(* IEC 61131-3 sources: RL_MAR/experiments/comparison/llm4plc/results/gpt-4o_20260507_114630/20260507_120848, 4 files *)

(* ---- generated_code_iteration_0.st ---- *)
plaintext
START_ST
FUNCTION_BLOCK FB_CourseDifferenceControl
VAR_INPUT
    KOMPASS_GRAD : INT; // Compass heading in tenths of a degree
    KURS         : INT; // Desired course in tenths of a degree
END_VAR
VAR_OUTPUT
    KURS_DIFF    : INT; // Computed course difference in tenths of a degree
END_VAR
VAR
    temp_diff    : INT; // Temporary variable for intermediate calculations
END_VAR

// Logic for course difference computation
IF KOMPASS_GRAD < 0 THEN
    KURS_DIFF := 0; // Set output to 0 if KOMPASS_GRAD is less than 0
ELSE
    temp_diff := KURS - KOMPASS_GRAD; // Calculate the initial difference
    IF temp_diff > 1800 THEN
        KURS_DIFF := temp_diff - 3600; // Adjust if the difference is greater than 1800
    ELSIF temp_diff < -1800 THEN
        KURS_DIFF := temp_diff + 3600; // Adjust if the difference is less than -1800
    ELSE
        KURS_DIFF := temp_diff; // No adjustment needed
    END_IF;
END_IF;

END_FUNCTION_BLOCK

PROGRAM MAIN
VAR
    fbCourseDifferenceControl : FB_CourseDifferenceControl; // Instance of the function block
    KOMPASS_GRAD_MAIN         : INT; // Compass heading input
    KURS_MAIN                 : INT; // Desired course input
    KURS_DIFF_MAIN            : INT; // Output course difference
END_VAR

// Initialize input variables
KOMPASS_GRAD_MAIN := 0; // Example initialization, can be replaced with actual values
KURS_MAIN := 0;         // Example initialization, can be replaced with actual values

// Call the function block
fbCourseDifferenceControl(KOMPASS_GRAD := KOMPASS_GRAD_MAIN, KURS := KURS_MAIN);

// Retrieve the output from the function block
KURS_DIFF_MAIN := fbCourseDifferenceControl.KURS_DIFF;

END_PROGRAM
END_ST

(* ---- generated_code_iteration_1.st ---- *)
START_REASON
The validation feedback indicates that the `MAIN` program cannot be instantiated in CODESYS. This error occurs because in Structured Text (ST), a `PROGRAM` type cannot be instantiated like a `FUNCTION_BLOCK`. Instead, the `PROGRAM` type is executed directly as part of the PLC cycle. The issue arises from attempting to create an instance of the `MAIN` program, which is not allowed.

To resolve this, the `PROGRAM MAIN` section should be modified to directly execute the logic without attempting to instantiate it. The `FUNCTION_BLOCK FB_CourseDifferenceControl` is correctly implemented and can be used within the `PROGRAM MAIN` by directly invoking its logic.

Additionally, the initialization of input variables and the retrieval of output variables should be adjusted to align with the corrected structure.

END_REASON

START_ST
FUNCTION_BLOCK FB_CourseDifferenceControl
VAR_INPUT
    KOMPASS_GRAD : INT; // Compass heading in tenths of a degree
    KURS         : INT; // Desired course in tenths of a degree
END_VAR
VAR_OUTPUT
    KURS_DIFF    : INT; // Computed course difference in tenths of a degree
END_VAR
VAR
    temp_diff    : INT; // Temporary variable for intermediate calculations
END_VAR

// Logic for course difference computation
IF KOMPASS_GRAD < 0 THEN
    KURS_DIFF := 0; // Set output to 0 if KOMPASS_GRAD is less than 0
ELSE
    temp_diff := KURS - KOMPASS_GRAD; // Calculate the initial difference
    IF temp_diff > 1800 THEN
        KURS_DIFF := temp_diff - 3600; // Adjust if the difference is greater than 1800
    ELSIF temp_diff < -1800 THEN
        KURS_DIFF := temp_diff + 3600; // Adjust if the difference is less than -1800
    ELSE
        KURS_DIFF := temp_diff; // No adjustment needed
    END_IF;
END_IF;

END_FUNCTION_BLOCK

PROGRAM MAIN
VAR
    fbCourseDifferenceControl : FB_CourseDifferenceControl; // Instance of the function block
    KOMPASS_GRAD_MAIN         : INT; // Compass heading input
    KURS_MAIN                 : INT; // Desired course input
    KURS_DIFF_MAIN            : INT; // Output course difference
END_VAR

// Initialize input variables
KOMPASS_GRAD_MAIN := 0; // Example initialization, can be replaced with actual values
KURS_MAIN := 0;         // Example initialization, can be replaced with actual values

// Call the function block
fbCourseDifferenceControl.KOMPASS_GRAD := KOMPASS_GRAD_MAIN;
fbCourseDifferenceControl.KURS := KURS_MAIN;
fbCourseDifferenceControl();

// Retrieve the output from the function block
KURS_DIFF_MAIN := fbCourseDifferenceControl.KURS_DIFF;

END_PROGRAM
END_ST

(* ---- generated_code_iteration_2.st ---- *)
START_REASON
The validation feedback indicates that the `PROGRAM MAIN` section contains an error because it attempts to instantiate the `MAIN` program, which is not allowed in CODESYS. In Structured Text (ST), a `PROGRAM` type is executed directly as part of the PLC cycle and cannot be instantiated like a `FUNCTION_BLOCK`.

To resolve this issue, the logic within the `PROGRAM MAIN` should directly execute the required functionality without attempting to create an instance of itself. The function block `FB_CourseDifferenceControl` is correctly implemented and can be used within the `PROGRAM MAIN` by directly invoking its logic.

Additionally, the initialization of input variables and the retrieval of output variables should be adjusted to align with the corrected structure. The corrected code will ensure proper execution without violating the rules of CODESYS.

END_REASON

START_ST
FUNCTION_BLOCK FB_CourseDifferenceControl
VAR_INPUT
    KOMPASS_GRAD : INT; // Compass heading in tenths of a degree
    KURS         : INT; // Desired course in tenths of a degree
END_VAR
VAR_OUTPUT
    KURS_DIFF    : INT; // Computed course difference in tenths of a degree
END_VAR
VAR
    temp_diff    : INT; // Temporary variable for intermediate calculations
END_VAR

// Logic for course difference computation
IF KOMPASS_GRAD < 0 THEN
    KURS_DIFF := 0; // Set output to 0 if KOMPASS_GRAD is less than 0
ELSE
    temp_diff := KURS - KOMPASS_GRAD; // Calculate the initial difference
    IF temp_diff > 1800 THEN
        KURS_DIFF := temp_diff - 3600; // Adjust if the difference is greater than 1800
    ELSIF temp_diff < -1800 THEN
        KURS_DIFF := temp_diff + 3600; // Adjust if the difference is less than -1800
    ELSE
        KURS_DIFF := temp_diff; // No adjustment needed
    END_IF;
END_IF;

END_FUNCTION_BLOCK

PROGRAM MAIN
VAR
    KOMPASS_GRAD_MAIN : INT; // Compass heading input
    KURS_MAIN         : INT; // Desired course input
    KURS_DIFF_MAIN    : INT; // Output course difference
    fbCourseDifferenceControl : FB_CourseDifferenceControl; // Instance of the function block
END_VAR

// Initialize input variables
KOMPASS_GRAD_MAIN := 0; // Example initialization, can be replaced with actual values
KURS_MAIN := 0;         // Example initialization, can be replaced with actual values

// Call the function block
fbCourseDifferenceControl.KOMPASS_GRAD := KOMPASS_GRAD_MAIN;
fbCourseDifferenceControl.KURS := KURS_MAIN;
fbCourseDifferenceControl();

// Retrieve the output from the function block
KURS_DIFF_MAIN := fbCourseDifferenceControl.KURS_DIFF;

END_PROGRAM
END_ST

(* ---- generated_code_iteration_3.st ---- *)
START_REASON
The validation feedback indicates that the `PROGRAM MAIN` section contains an error because it attempts to instantiate the `MAIN` program, which is not allowed in CODESYS. In CODESYS, a `PROGRAM` type cannot be instantiated like a `FUNCTION_BLOCK`. Instead, the logic within the `PROGRAM MAIN` should directly execute the required functionality without attempting to create an instance of itself.

To resolve this issue, the instantiation of the `fbCourseDifferenceControl` function block within the `PROGRAM MAIN` should be removed. Instead, the logic of the function block should be invoked directly within the program. The corrected code will ensure proper execution without violating the rules of CODESYS.

END_REASON

START_ST
FUNCTION_BLOCK FB_CourseDifferenceControl
VAR_INPUT
    KOMPASS_GRAD : INT; // Compass heading in tenths of a degree
    KURS         : INT; // Desired course in tenths of a degree
END_VAR
VAR_OUTPUT
    KURS_DIFF    : INT; // Computed course difference in tenths of a degree
END_VAR
VAR
    temp_diff    : INT; // Temporary variable for intermediate calculations
END_VAR

// Logic for course difference computation
IF KOMPASS_GRAD < 0 THEN
    KURS_DIFF := 0; // Set output to 0 if KOMPASS_GRAD is less than 0
ELSE
    temp_diff := KURS - KOMPASS_GRAD; // Calculate the initial difference
    IF temp_diff > 1800 THEN
        KURS_DIFF := temp_diff - 3600; // Adjust if the difference is greater than 1800
    ELSIF temp_diff < -1800 THEN
        KURS_DIFF := temp_diff + 3600; // Adjust if the difference is less than -1800
    ELSE
        KURS_DIFF := temp_diff; // No adjustment needed
    END_IF;
END_IF;

END_FUNCTION_BLOCK

PROGRAM MAIN
VAR
    KOMPASS_GRAD_MAIN : INT; // Compass heading input
    KURS_MAIN         : INT; // Desired course input
    KURS_DIFF_MAIN    : INT; // Output course difference
END_VAR

// Initialize input variables
KOMPASS_GRAD_MAIN := 0; // Example initialization, can be replaced with actual values
KURS_MAIN := 0;         // Example initialization, can be replaced with actual values

// Logic for course difference computation using FB_CourseDifferenceControl
IF KOMPASS_GRAD_MAIN < 0 THEN
    KURS_DIFF_MAIN := 0; // Set output to 0 if KOMPASS_GRAD_MAIN is less than 0
ELSE
    VAR temp_diff : INT; // Temporary variable for intermediate calculations
    temp_diff := KURS_MAIN - KOMPASS_GRAD_MAIN; // Calculate the initial difference
    IF temp_diff > 1800 THEN
        KURS_DIFF_MAIN := temp_diff - 3600; // Adjust if the difference is greater than 1800
    ELSIF temp_diff < -1800 THEN
        KURS_DIFF_MAIN := temp_diff + 3600; // Adjust if the difference is less than -1800
    ELSE
        KURS_DIFF_MAIN := temp_diff; // No adjustment needed
    END_IF;
END_IF;

END_PROGRAM
END_ST
